{attribute 'TcGenerated'}
{attribute 'no-analysis'}
{attribute 'linkalways'}
// This function has been automatically generated from the project information.
VAR_GLOBAL CONSTANT
	{attribute 'const_non_replaced'}
	stLibVersion_Tk_Diagnosis_IO_LinkMaster : ST_LibVersion := (iMajor := 0, iMinor := 0, iBuild := 2, iRevision := 1, nFlags := 0, sVersion := '0.0.2.1');
END_VAR

(* stored: Version 1.1.0.1
   GVL Global_Version: Id {9a7a2ece-fcca-447f-8f80-dd4adb9d5376} *)
